{attribute 'qualified_only'}
TYPE E_Brightness :
(
	high :=16#00,
    medium :=16#01,
    low :=16#02
) INT;
END_TYPE

(* stored: Version 1.1.0.1, ProductVersion 3.1.4024.9
   DUT E_Brightness: Id {ef0f1782-cdba-4576-b48a-8ea3e5a71bfc} *)
